{attribute addProperty BoxType "EL6201-0000-0017"}
{attribute addProperty Id "Slave_29A_DI0BIT10.125225Slave_29A_DI1BIT10.125226Slave_29A_DI2BIT10.125227Slave_29A_DI3BIT10.125228Slave_29B_DI0BIT10.125229Slave_29B_DI1BIT10.125230Slave_29B_DI2BIT10.125231Slave_29B_DI3BIT10.125232"}
{attribute addProperty CRC "2408794620"}
{attribute addProperty SizeInBites "8"}
{attribute addProperty SizeInBytes "1"}
TYPE Slave_29_Inputs_8F9349FC :
STRUCT
	{attribute addProperty Name "Slave_29A_DI0"}
	Slave_29A_DI0 : BIT;
	{attribute addProperty Name "Slave_29A_DI1"}
	Slave_29A_DI1 : BIT;
	{attribute addProperty Name "Slave_29A_DI2"}
	Slave_29A_DI2 : BIT;
	{attribute addProperty Name "Slave_29A_DI3"}
	Slave_29A_DI3 : BIT;
	{attribute addProperty Name "Slave_29B_DI0"}
	Slave_29B_DI0 : BIT;
	{attribute addProperty Name "Slave_29B_DI1"}
	Slave_29B_DI1 : BIT;
	{attribute addProperty Name "Slave_29B_DI2"}
	Slave_29B_DI2 : BIT;
	{attribute addProperty Name "Slave_29B_DI3"}
	Slave_29B_DI3 : BIT;
END_STRUCT
END_TYPE

(* stored: Version 1.2.0.0, ProductVersion 3.1.4024.9
   DUT Slave_29_Inputs_8F9349FC: Id {da2a367f-8593-42f5-93f1-fde3d4da25cd} *)
